// TIA Portal V18 export
FUNCTION_BLOCK "Display_management"   // FB7, LAD
{ S7_Optimized_Access := 'TRUE' }
VERSION : 0.1
// stored: AutoNumber true, IsIECCheckEnabled false, IsRetainMemResEnabled false, MemoryReserve 100, SetENOAutomatically false, UDAEnableTagReadback false
   VAR_TEMP   // added for the SCL form of the ladder/FBD networks
      _w1 : Bool;
      _w2 : Bool;
   END_VAR
BEGIN

REGION Network 1: reseting the Quantity, HSC
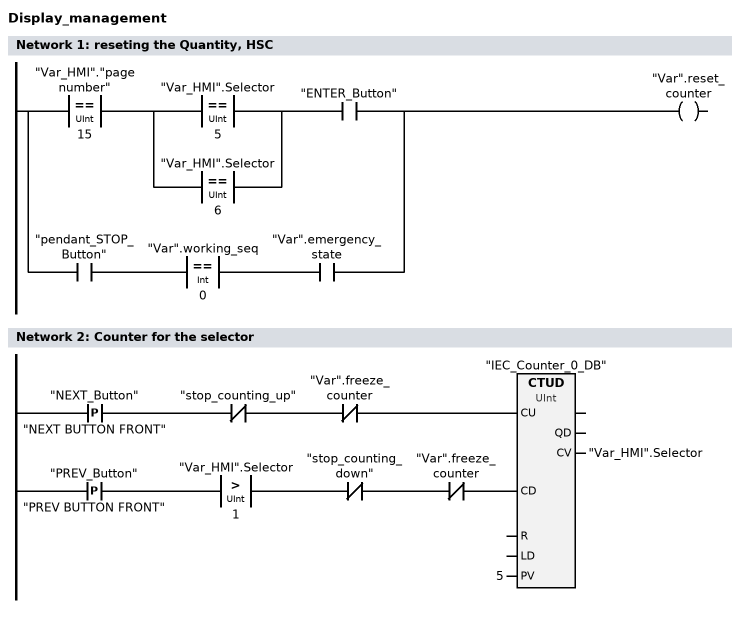
   RUNG wire#powerrail
      { S7_Templates := "SrcType := UInt" } EQ_Contact(in1 := "Var_HMI"."page number", in2 := 15)
      wire#w1
      { S7_Templates := "SrcType := UInt" } EQ_Contact(in1 := "Var_HMI".Selector, in2 := 5)
      wire#w2
      Contact( "ENTER_Button" )
      wire#w3
      Coil( "Var".reset_counter )
   END_RUNG
   RUNG wire#w1
      { S7_Templates := "SrcType := UInt" } EQ_Contact(in1 := "Var_HMI".Selector, in2 := 6)
   END_RUNG wire#w2
   RUNG wire#powerrail
      Contact( "pendant_STOP_Button" )
      { S7_Templates := "SrcType := Int" } EQ_Contact(in1 := "Var".working_seq, in2 := 0)
      Contact( "Var".emergency_state )
   END_RUNG wire#w3
   // the same network as SCL:
   "Var".reset_counter := (("Var_HMI"."page number" = 15) AND (("Var_HMI".Selector = 5) OR ("Var_HMI".Selector = 6)) AND "ENTER_Button") OR ("pendant_STOP_Button" AND ("Var".working_seq = 0) AND "Var".emergency_state);
END_REGION

REGION Network 2: Counter for the selector
   RUNG wire#powerrail
      P_Contact(operand := "NEXT_Button", bit := "NEXT BUTTON FRONT")
      I_Contact( "stop_counting_up" )
      I_Contact( "Var".freeze_counter )
      { S7_Templates := "value_type := UInt" } "IEC_Counter_0_DB".CTUD(cd := wire#w1, r :=, ld :=, pv := 5, qd =>, cv => "Var_HMI".Selector)
   END_RUNG
   RUNG wire#powerrail
      P_Contact(operand := "PREV_Button", bit := "PREV BUTTON FRONT")
      { S7_Templates := "SrcType := UInt" } GT_Contact(in1 := "Var_HMI".Selector, in2 := 1)
      I_Contact( "stop_counting_down" )
      I_Contact( "Var".freeze_counter )
   END_RUNG wire#w1
   // the same network as SCL:
   #_w1 := "NEXT_Button" AND NOT "NEXT BUTTON FRONT";   // rising edge of "NEXT_Button"
   "NEXT BUTTON FRONT" := "NEXT_Button";
   #_w2 := "PREV_Button" AND NOT "PREV BUTTON FRONT";   // rising edge of "PREV_Button"
   "PREV BUTTON FRONT" := "PREV_Button";
   "IEC_Counter_0_DB".CTUD(CU := #_w1 AND NOT "stop_counting_up" AND NOT "Var".freeze_counter,
                           CD := #_w2 AND ("Var_HMI".Selector > 1) AND NOT "stop_counting_down" AND NOT "Var".freeze_counter,
                           PV := 5,
                           CV => "Var_HMI".Selector);
END_REGION

REGION Network 3 (SCL): Condition for reseting the Menu counter
   IF     ("Var_HMI"."page number"=12 AND "Var_HMI".Selector>5)
       OR ("Var_HMI"."page number"=13 AND "Var_HMI".Selector>6)
       OR ("Var_HMI"."page number"=14 AND "Var_HMI".Selector>3)
       OR ("Var_HMI"."page number"=15 AND "Var_HMI".Selector>5)
       OR ("Var_HMI"."page number"=18 AND "Var_HMI".Selector>3)
       OR ("Var_HMI"."page number"=20 AND "Var_HMI".Selector>4)
       OR ("Var_HMI"."page number"=21 AND "Var_HMI".Selector>4)
       OR ("Var_HMI"."page number"=23 AND "Var_HMI".Selector>5)
       OR ("Var_HMI"."page number"=24 AND "Var_HMI".Selector>4)
       OR ("Var_HMI"."page number"=14 AND "Var_HMI".Selector>8)
       OR ("Var_HMI"."page number"=30 AND "Var_HMI".Selector>8)
       OR ("Var_HMI"."page number"=40 AND "Var_HMI".Selector>7)
   THEN
       "stop_counting_up" := 1;
   ELSE
       "stop_counting_up" := 0;
   END_IF;

   //Limitation for selector (OP fault prevetion)
   IF "Var_HMI"."page number" = 15 AND "Var_HMI".Selector<=5 THEN
       "stop_counting_down" := 1;
   ELSE
       "stop_counting_down" := 0;
   END_IF;


           // To freeze the counter
   "Var".freeze_counter := "Var".working_seq = 10
   OR "Var_HMI".in_selection
   OR "Var".emergency_flag
   OR "Var".pause_flag
   OR "Var".draining_flag
   OR ("Var_HMI"."page number" = 18);
END_REGION

REGION Network 4 (SCL): Page selector, for the Template icons

   //page12
   IF  "Var_HMI".Selector = 1 AND "Rising_edge_enter".Q THEN
       "Rising_edge_enter".Q := 0;
       "Var_HMI"."page number" := 12;
   END_IF;


   //page 20
   IF ("Var_HMI".Selector = 2 AND "Rising_edge_enter".Q) THEN
       "Rising_edge_enter".Q:= 0;
       "IEC_Counter_0_DB".CV := 5;
       "Var_HMI"."page number" := 20;

   END_IF;

   //page 20
   IF "Var_HMI"."page number" = 20 THEN

       IF "Var_HMI".Selector = 5 AND "Rising_edge_enter".Q THEN
           "IEC_Counter_0_DB".CV := 5;
           "Rising_edge_enter".Q:= 0;
           "Var_HMI"."page number" := 21;
       END_IF;

   END_IF;

   //page 21
   IF "Var_HMI"."page number" = 21 THEN

       IF "Var_HMI".Selector = 5 AND "Rising_edge_enter".Q THEN
           "Rising_edge_enter".Q := 0;
           "Var_HMI"."page number" := 20;
       END_IF;

   END_IF;

   //page 30
   IF ("Var_HMI".Selector = 3 AND "Rising_edge_enter".Q) THEN
       "Rising_edge_enter".Q := 0;
       "Var_HMI"."page number" := 30;
   END_IF;


   //page 40
   IF ("Var_HMI".Selector = 4 AND "Rising_edge_enter".Q) THEN
       "Rising_edge_enter".Q := 0;
       "Var_HMI"."page number" := 40;
   END_IF;
END_REGION

REGION Network 5 (SCL): Page 12, HOME
   //some condition should be added

   IF "Var_HMI"."page number" = 12 AND "Var".emergency_state THEN

       //Loading
       IF "Var_HMI".Selector = 5 AND "Rising_edge_enter".Q THEN

           "Var".Total_quantity := 0;
           "Var".lotto_terminato := 0;
           "Rising_edge_enter".Q := 0; 
           "IEC_Counter_0_DB".CV := 5;
           "Var_HMI"."page number" := 13;


       END_IF;

       //Drain
       IF "Var_HMI".Selector = 6 AND "Rising_edge_enter".Q THEN

           "Rising_edge_enter".Q := 0;
           "IEC_Counter_0_DB".CV := 6;
           "Var_HMI"."page number" := 23;


       END_IF;



   END_IF;
END_REGION

REGION Network 6 (SCL): Page 13 Loading setup
   //some condition should be added
   IF "Var_HMI"."page number" = 13 AND "Var".emergency_state THEN


       //"Var".reset_counter := 0;
       "EDIT_SET_QUANTITY".TON(IN:="ENTER_Button",
                               PT:=T#2000ms);

       //Set Timer for 
       IF "Var_HMI".Selector = 5 AND "EDIT_SET_QUANTITY".Q THEN

           "Var_HMI"."selection_no" := 1;
           "Var_HMI".in_selection:=1;


       END_IF;

       //Flow rate th
       IF "Var_HMI".Selector = 6 AND "EDIT_SET_QUANTITY".Q THEN

           "Var_HMI"."selection_no" := 2;
           "Var_HMI".in_selection := 1;

       END_IF;

       IF "Var_HMI".Selector=7 AND "Pendant_START_Button" AND "Var".set_quantity>0 AND "Var".FCV_high_flow_signal>0 THEN

           "Var".In_loading := 1;
           "Var".In_Draining := 0;
           "Var_HMI"."page number" := 14; 

       END_IF;

   END_IF;

   IF NOT "ENTER_Button" THEN
       RESET_TIMER("EDIT_SET_QUANTITY");
   END_IF;
END_REGION

REGION Network 7 (SCL): Page 14 In Loading
   //The condition need to be checked
   IF "Var_HMI"."page number" = 14 AND "Var".loaded_quantity >= "Var".set_quantity THEN
       "IEC_Counter_0_DB".CV := 5;
       "Var".Number_of_IBC := "Var".Number_of_IBC + 1;
       "Var".Total_quantity := "Var".Total_quantity + "Var".loaded_quantity;
       "Var_HMI"."page number" := 15;



   END_IF;
END_REGION

REGION Network 8 (SCL): Page 15, Lotto terminato
   IF "Var_HMI"."page number" = 15 AND "Var".emergency_state THEN



       "Var".lotto_terminato := 0;  //check this because you're resetting at page 12 

       IF "Var_HMI".Selector = 5 AND "Rising_edge_enter".Q THEN

           "Rising_edge_enter".Q := 0;
           "Var_HMI"."page number" := 13;

       END_IF;


       IF "Var_HMI".Selector = 6 AND "Rising_edge_enter".Q THEN

           "Rising_edge_enter".Q := 0;
           "IEC_Counter_0_DB".CV := 5;
           "Var_HMI"."page number" := 18;
           "Var".lotto_terminato := 1;

       END_IF;


   END_IF;
END_REGION

REGION Network 9 (SCL): Page 18, RIPIELOGO TERMINATO
   IF "Var_HMI"."page number"=18  THEN

       "Var".In_loading := 0;
       "Var".In_Draining := 0;


       IF "Rising_edge_enter".Q THEN
           "Var_HMI"."page number" := 12;
           "Var".Total_quantity := 0;
           "Rising_edge_enter".Q := 0;
           "Var".No_of_IBC_all_time := "Var".No_of_IBC_all_time + "Var".Number_of_IBC;
           "Var".Number_of_IBC := 0;
       END_IF;




   END_IF;
END_REGION

REGION Network 10 (SCL): Page 20 and 21, IOs
   IF "Var_HMI"."page number" = 20 THEN

       IF "Var_HMI".Selector = 5 AND "Rising_edge_enter".Q THEN
           "Var_HMI"."page number" := 21;
           "Rising_edge_enter".Q := 0;
       END_IF;

   END_IF;

   IF "Var_HMI"."page number" = 21 THEN

       IF "Var_HMI".Selector = 5 AND "Rising_edge_enter".Q THEN
           "Var_HMI"."page number" := 20;
           "Rising_edge_enter".Q := 0;
       END_IF;

   END_IF;
END_REGION

REGION Network 11 (SCL): Page 23, Drain pages setting
   IF "Var_HMI"."page number" = 23 AND "Var".emergency_state THEN


       "IEC_Timer_0_DB_4".TON(IN := "ENTER_Button",
                              PT := T#2S);




       //(Set Time FOR the timer, is it needed?
       IF "Var_HMI".Selector = 5 AND "IEC_Timer_0_DB_4".Q THEN

           "Var_HMI"."selection_no" := 3;
           "Var_HMI".in_selection := 1;

       END_IF;


       IF "Var_HMI".Selector = 6 AND "Pendant_START_Button" THEN
           "Var".In_Draining := 1;
           "Var_HMI"."page number" := 24;
           "IEC_Counter_0_DB".CV := 5;
       END_IF;


   END_IF;
END_REGION

REGION Network 12 (SCL): Page 24 Drain page
   IF "Var_HMI"."page number" = 24 THEN

       IF "Var_HMI".Selector = 5 AND "Rising_edge_enter".Q AND NOT ("Var".emergency_flag OR "Var".pause_flag OR "Var".draining_flag)  THEN

           "Var".In_Draining := 0;
           "Rising_edge_enter".Q := 0;
           "Var_HMI"."page number" := 12;
       END_IF;

   END_IF;
END_REGION

REGION Network 13 (SCL): Page 30, settings and default values


   IF "Var_HMI"."page number" = 30 THEN

       "IEC_Timer_0_DB_12".TON(IN:="ENTER_Button",
                               PT:=T#1500ms);




       IF "Var_HMI".Selector = 5 AND "IEC_Timer_0_DB_12".Q THEN
           "Var_HMI".selection_no := 8;
           "Var_HMI".in_selection := 1;


       END_IF;

       IF "Var_HMI".Selector = 6 AND "IEC_Timer_0_DB_12".Q THEN
           "Var_HMI".selection_no := 9;
           "Var_HMI".in_selection := 1;


       END_IF;

       IF "Var_HMI".Selector = 7 AND "IEC_Timer_0_DB_12".Q THEN
           "Var_HMI".selection_no := 10;
           "Var_HMI".in_selection := 1;


       END_IF;

       IF "Var_HMI".Selector = 8 AND "IEC_Timer_0_DB_12".Q THEN
           "Var_HMI".selection_no := 11;
           "Var_HMI".in_selection := 1;
           "Rising_edge_enter".Q := 0;

       END_IF;

       IF "Var_HMI".Selector = 9 AND "IEC_Timer_0_DB_12".Q THEN
           "Var_HMI".selection_no := 12;
           "Var_HMI".in_selection := 1;
           "Rising_edge_enter".Q := 0;
       END_IF;






   END_IF;

   IF NOT "ENTER_Button" THEN

       RESET_TIMER("IEC_Timer_0_DB_12");

   END_IF;
END_REGION

REGION Network 14 (SCL): page 40
   IF "Var_HMI"."page number" = 40 THEN

       "Scrolling_1_Timer".TON(IN := "ENTER_Button",
                               PT := T#1.5S);


       IF "Var_HMI".Selector = 5 AND "Scrolling_1_Timer".Q THEN

           "Var_HMI"."selection_no" := 4;
           "Var_HMI".in_selection := 1;


       END_IF;


       IF "Var_HMI".Selector = 6 AND "Scrolling_1_Timer".Q THEN

           "Var_HMI"."selection_no" := 5;
           "Var_HMI".in_selection := 1;

       END_IF;

      IF "Var_HMI".Selector = 7 AND "Scrolling_1_Timer".Q THEN

           "Var_HMI"."selection_no" := 6;
           "Var_HMI".in_selection := 1;

       END_IF;


       IF "Var_HMI".Selector = 8 AND "Scrolling_1_Timer".Q THEN

           "Var_HMI"."selection_no" := 7;
           "Var_HMI".in_selection := 1;
       END_IF;

   END_IF;
END_REGION

REGION Network 15 (SCL): In_Selection handling
   IF "Var_HMI".in_selection THEN

       CASE "Var_HMI".selection_no OF



           //Set Quantity       
           1:

                 "IEC_Timer_0_DB".TP(IN:="Clock_10Hz",
                                     PT:=T#0.001s);

                 IF "IEC_Timer_0_DB".Q THEN


                     IF "NEXT_Button" THEN
                         "Var".set_quantity := "Var".set_quantity + 10;
                     END_IF;


                     IF "PREV_Button" THEN
                         "Var".set_quantity := "Var".set_quantity - 10;
                         "Var".set_quantity := MAX(IN1 := "Var".set_quantity, IN2 := 0);


                     END_IF;


                     IF "ENTER_Button" THEN
                         "Var_HMI".in_selection := 0;
                         "Var_HMI".selection_no := 0;

                     END_IF;


                 END_IF;

                 ;





               //Set Flowrate
           2:

               "IEC_Timer_0_DB_1".TP(IN:="Clock_10Hz",
                                     PT:=T#0.001s);

               IF "IEC_Timer_0_DB_1".Q THEN


                   IF "NEXT_Button" THEN
                       "Var".FCV_high_flow_signal := "Var".FCV_high_flow_signal + 1;
                   END_IF;

                   IF "PREV_Button" THEN
                       "Var".FCV_high_flow_signal := "Var".FCV_high_flow_signal - 1;
                       "Var".FCV_high_flow_signal := MAX(IN1 := "Var".FCV_high_flow_signal, IN2 := 0);
                   END_IF;

                   IF "ENTER_Button" THEN
                       "Var_HMI".in_selection := 0;
                       "Var_HMI".selection_no := 0;
                   END_IF;

               END_IF;

               ;




               //Draining time
           3:


               "IEC_Timer_0_DB_2".TP(IN := "Clock_10Hz",
                                     PT := T#0.01s);

               IF "IEC_Timer_0_DB_2".Q THEN

                   IF "NEXT_Button" THEN
                       "Var".drain_time_integer := "Var".drain_time_integer + 100;
                       "Var".drain_time_integer_seconds := ROUND(IN := "Var".drain_time_integer / 1000);

                   END_IF;

                   IF "PREV_Button" THEN
                       "Var".drain_time_integer := "Var".drain_time_integer - 100;
                       "Var".drain_time_integer_seconds := ROUND(IN := "Var".drain_time_integer / 1000);
                       "Var".drain_time_integer_seconds := MAX(IN1 := "Var".drain_time_integer_seconds, IN2 := 0);
                       END_IF;

                   IF "ENTER_Button" THEN
                       "Var".drain_time_time := INT_TO_TIME(IN := "Var".drain_time_integer);
                       "Var_HMI"."in_selection" := 0;
                       "Var_HMI".selection_no := 0;
                   END_IF;


               END_IF;

               ;




               //scrolling 1
                   4:

                   "IEC_Timer_0_DB_6".TP(IN:="Clock_10Hz",
                                         PT:=T#0.001S);
                   IF NOT "ENTER_Button" THEN

                       "Scrolling_1_Timer".IN := FALSE;
                       "Var_HMI".in_selection := 0;
                       "Var_HMI".selection_no := 0;
                   END_IF;

                   IF "IEC_Timer_0_DB_6".Q AND "Var_HMI".in_selection  THEN

                       IF "ENTER_Button" THEN
                           "Var_HMI".scrolling_1 := "Var_HMI".scrolling_1 - 1;
                           "Var_HMI".scrolling_1 := MAX(IN1 := "Var_HMI".scrolling_1, IN2 := 0);
                       END_IF;

                   END_IF;

                   ;




                   //scrolling 2
           5:

               "IEC_Timer_0_DB_7".TP(IN := "Clock_10Hz",
                                     PT := T#0.001S);

               IF NOT "ENTER_Button" THEN

                   "Scrolling_1_Timer".IN := FALSE;
                   "Var_HMI".in_selection := 0;
                   "Var_HMI".selection_no := 0;
               END_IF;

               IF "IEC_Timer_0_DB_7".Q AND "Var_HMI".in_selection THEN

                   IF "ENTER_Button" THEN
                       "Var_HMI".scrolling_1 := "Var_HMI".scrolling_1 + 1;
                       "Var_HMI".scrolling_1 := MAX(IN1 := "Var_HMI".scrolling_1, IN2 := 0);
                   END_IF;

               END_IF;





               //scrolling 3
           6:

               "IEC_Timer_0_DB_8".TP(IN:="Clock_1Hz",
                                     PT:=T#0.001s);



               IF NOT "ENTER_Button" THEN

                   "Scrolling_1_Timer".IN := FALSE;
                   "Var_HMI".in_selection := 0;
                   "Var_HMI".selection_no := 0;
               END_IF;

               IF "IEC_Timer_0_DB_8".Q AND "Var_HMI".in_selection THEN

                   IF "ENTER_Button" THEN
                       "Var_HMI".scrolling_2 := "Var_HMI".scrolling_2 - 1;
                       "Var_HMI".scrolling_2 := MAX(IN1 := "Var_HMI".scrolling_2, IN2 := 0);
                   END_IF;

               END_IF;






               //scrolling 4 
           7:

               "IEC_Timer_0_DB_9".TP(IN:="Clock_1Hz",
                                     PT:=T#0.001s);



               IF NOT "ENTER_Button" THEN

                   "Scrolling_1_Timer".IN := FALSE;
                   "Var_HMI".in_selection := 0;
                   "Var_HMI".selection_no := 0;
               END_IF;

               IF "IEC_Timer_0_DB_9".Q AND "Var_HMI".in_selection THEN

                   IF "ENTER_Button" THEN
                       "Var_HMI".scrolling_2 := "Var_HMI".scrolling_2 + 1;
                   END_IF;

               END_IF;





               // Set the default Quantity
           8:

                  "IEC_Timer_0_DB_14".TP(IN:="Clock_10Hz",
                                         PT:=T#0.001s);
                  IF "IEC_Timer_0_DB_14".Q THEN

                  IF "NEXT_Button" THEN
                      "Var".set_quantity := "Var".set_quantity + 10;
                  END_IF;

                  IF "PREV_Button" THEN
                      "Var".set_quantity := "Var".set_quantity - 10;
                      "Var".set_quantity := MAX(IN1 := "Var".set_quantity, IN2 := 0);



                  END_IF;

                  IF "ENTER_Button" THEN
                      "Var_HMI".in_selection := 0;
                      "Var_HMI".selection_no := 0;


                  END_IF;
              END_IF;

               ;




               //Set the default flowrate
           9:
              "IEC_Timer_0_DB_17".TP(IN:="Clock_10Hz",
                                     PT:=T#0.001s);

              IF "IEC_Timer_0_DB_17".Q THEN

                  IF "NEXT_Button" THEN
                      "Var".FCV_high_flow_signal := "Var".FCV_high_flow_signal + 10;
                  END_IF;

                  IF "PREV_Button" THEN
                      "Var".FCV_high_flow_signal := "Var".FCV_high_flow_signal - 10;
                      "Var".FCV_high_flow_signal := MAX(IN1 := "Var".FCV_high_flow_signal, IN2 := 0);
                  END_IF;

                  IF "ENTER_Button" THEN

                      "Var_HMI".in_selection := 0;
                      "Var_HMI".selection_no := 0;


                  END_IF;

              END_IF;
               ;





               // Set default initial low flowrate percentage quantity
           10:


                   IF "Rising_edge_next".Q THEN
                       "Var".quantity_of_LH_flow_percentage_initial := "Var".quantity_of_LH_flow_percentage_initial + 1;
                       "Rising_edge_next".Q:=0;
                   END_IF;

                   IF "Rising_edge_prev".Q THEN
                       "Var".quantity_of_LH_flow_percentage_initial := "Var".quantity_of_LH_flow_percentage_initial - 1;
                       "Var".quantity_of_LH_flow_percentage_initial := MAX(IN1 := "Var".quantity_of_LH_flow_percentage_initial, IN2 := 0);
                       "Rising_edge_prev".Q := 0;

                   END_IF;

                   IF "Rising_edge_enter".Q THEN
                       "Var_HMI".in_selection := 0;
                       "Var_HMI".selection_no := 0;
                       "Rising_edge_enter".Q := 0;
                   END_IF;


               ;



               // Set default initial low flowrate percentage quantity
           11:

                   IF "Rising_edge_next".Q THEN
                       "Var".quantity_of_HL_flow_percentage_final := "Var".quantity_of_HL_flow_percentage_final + 1;
                       "Rising_edge_next".Q := 0;
                   END_IF;

                   IF "Rising_edge_prev".Q THEN
                       "Var".quantity_of_HL_flow_percentage_final := "Var".quantity_of_HL_flow_percentage_final - 1;
                       "Var".quantity_of_HL_flow_percentage_final := MAX(IN1 := "Var".quantity_of_HL_flow_percentage_final, IN2 := 0);
                       "Rising_edge_prev".Q := 0;
                   END_IF;

                   IF "Rising_edge_enter".Q THEN
                       "Var_HMI".in_selection := 0;
                       "Var_HMI".selection_no := 0;
                       "Rising_edge_enter".Q := 0;
                   END_IF;



               ;




               // Set default initial low flowrate percentage quantity
           12:
               "IEC_Timer_0_DB_16".TP(IN := "Clock_10Hz",
                                      PT := T#0.001S);
               IF "IEC_Timer_0_DB_16".Q THEN
                   IF "NEXT_Button" THEN
                       "Var".FCV_low_flow_signal:= "Var".FCV_low_flow_signal + 100;
                   END_IF;

                   IF "PREV_Button" THEN
                       "Var".FCV_low_flow_signal := "Var".FCV_low_flow_signal - 100;
                       "Var".FCV_low_flow_signal := MAX(IN1 := "Var".FCV_low_flow_signal, IN2 := 0);
                   END_IF;

                   IF "ENTER_Button" THEN
                       "Var_HMI".in_selection := 0;
                       "Var_HMI".selection_no := 0;

                   END_IF;

               END_IF;


               ;

       END_CASE;
   END_IF;
END_REGION

REGION Network 16 (SCL): Emergency Handling
   IF "Var".emergency_state AND "Var_HMI".emergency_popup AND "ENTER_Button" THEN

       "Var_HMI".emergency_popup := 0;

   END_IF;
END_REGION
END_FUNCTION_BLOCK
